Fanuc TP program (LS listing): _FLTOVC.LS

/PROG  _FLTOVC
/ATTR
OWNER		= MNEDITOR;
COMMENT		= "Over Current Alm";
PROG_SIZE	= 298;
CREATE		= DATE 21-03-19  TIME 11:14:44;
MODIFIED	= DATE 21-03-19  TIME 11:14:44;
FILE_NAME	= _FLTCOL;
VERSION		= 0;
LINE_COUNT	= 4;
MEMORY_SIZE	= 662;
PROTECT		= READ_WRITE;
TCD:  STACK_SIZE	= 0,
      TASK_PRIORITY	= 50,
      TIME_SLICE	= 0,
      BUSY_LAMP_OFF	= 0,
      ABORT_REQUEST	= 0,
      PAUSE_REQUEST	= 0;
DEFAULT_GROUP	= *,*,*,*,*;
CONTROL_CODE	= 00000000 00000000;
/APPL
/APPL
/MN
   1:  !***************************** ;
   2:  !Over Current Alarm ;
   3:  !***************************** ;
   4:  CALL _FAULT(14) ;
/POS
/END
